(* IEC 61131-3 sources: programs/VI-54/VI-54_20171205/VI-54_20171205/Stations/Screen/LseClass170718/Class/WindowEnd, 1 file *)

(* ---- WindowEnd.st ---- *)
(*!
<Class
	Name               = "WindowEnd"
	Revision           = "0.0"
	RealtimeTask       = "false"
	CyclicTask         = "false"
	BackgroundTask     = "false"
	Sigmatek           = "false"
	OSInterface        = "false"
	HighPriority       = "false"
	Automatic          = "false"
	UpdateMode         = "Prescan"
	SharedCommandTable = "true"
	Objectsize         = "(284,120)">
	<Channels>
	</Channels>
	<Network Name="WindowEnd">
		<!-- List of Components in this network -->
		<Components>
			<Object
				Name       = "_base"
				Class      = "_Global"
				Position   = "(218,120)"
				Visualized = "true"
				Remotely   = "true">
				<Channels>
					<Server Name="Server0">
						<OPCSettings WriteProtected="false"/>
					</Server>
					<Client Name="Lse"/>
				</Channels>
			</Object>
		</Components>
		<Comments>
		</Comments>
		<!-- List of Connections in this network -->
		<Connections>
			<Connection Source="this.Server0" Destination="_base.Server0" Vertices="(690,210),(518,210),"/>
			<Connection Source="_base.Lse" Destination="this.Lse" Vertices="(218,210),(38,210),"/>
		</Connections>
		<!-- Headerfiles -->
		<Options>
		</Options>
	</Network>
</Class>
*)
#pragma using _Global

WindowEnd : CLASS
: _Global
  //Servers:
  //Clients:
  //Variables:
		WindowClose 	: DINT;
  //Functions:

	FUNCTION VIRTUAL GLOBAL IF_WindowEnd
		VAR_INPUT
			whoami 	: ^_WHOAMI;
			pic 	: ^void;
		END_VAR;

	FUNCTION GLOBAL Read_WindowEnd
		VAR_INPUT
			Reset 	: DINT;
		END_VAR
		VAR_OUTPUT
			End 	: DINT;
		END_VAR;
  //Tables:
	FUNCTION @STD
		VAR_OUTPUT
			ret_code	: CONFSTATES;
		END_VAR;
	FUNCTION GLOBAL TAB @CT_;
END_CLASS;

FUNCTION VIRTUAL GLOBAL WindowEnd::IF_WindowEnd
	VAR_INPUT
		whoami 	: ^_WHOAMI;
		pic 	: ^void;
	END_VAR

  WindowClose := 1;

END_FUNCTION

FUNCTION GLOBAL WindowEnd::Read_WindowEnd
	VAR_INPUT
		Reset 	: DINT;
	END_VAR
	VAR_OUTPUT
		End 	: DINT;
	END_VAR

  if Reset = 1 then
    WindowClose := 0;
  else
    End := WindowClose;
  end_if;

END_FUNCTION
